Fanuc KAREL source: kf00111.KL

PROGRAM KF00111
%STACKSIZE=65535
%PRIORITY=65535
%NOLOCKGROUP
VAR
I : INTEGER
J : INTEGER
X : REAL
Y : REAL
B : BOOLEAN
C : BOOLEAN
TXT : STRING[80]
TXT2 : STRING[80]
AI : ARRAY[4] OF INTEGER
BI : ARRAY[4] OF INTEGER
P : XYZWPR
JP : JOINTPOS9
PF : POSITION
STATUS : INTEGER
-- UNRESOLVED DECLARATIONS (source type spelling not recovered)
-- V1 : TYPE_0x0013 (type_u16=0x0013)
-- V2 : TYPE_0x0013 (type_u16=0x0013)
BEGIN
I=1
X=1.0
B=TRUE
-- UNSAFE_SOURCE_IR line 24: X = int_to_real(native_io_value(3, 1))
END KF00111
